(* IEC 61131-3 sources: RAG_PLC/data/result/test/022, 2 files *)

(* ---- wrapped.st ---- *)
(* =========================================================
   Generated by PLC-Eval Benchmark Wrapper
   ========================================================= *)

FUNCTION_BLOCK LLM_Wrapper_FB
PROGRAM Main
VAR
    StartChk : BOOL;
    Regen : BOOL;
    ErrorFlag : BOOL;
END_VAR

// Step 1: Start Check
IF NOT StartChk THEN
    StartChk := TRUE;
    // Additional initialization code here
END_IF;

// Step 2: Regeneration Check
IF StartChk AND NOT Regen THEN
    Regen := TRUE;
    // Additional regeneration code here
END_IF;

// Error Handling
IF ErrorFlag THEN
    // Stop program
    // Issue error message to visualization system
    // Additional error handling code here
END_IF;

END_PROGRAM
END_FUNCTION_BLOCK

PROGRAM Auto_Proxy_Prg
  VAR
    instance : LLM_Wrapper_FB;
  END_VAR

  instance();
END_PROGRAM

CONFIGURATION Config0
  RESOURCE Res0 ON PLC
    TASK TaskMain(INTERVAL := T#20ms, PRIORITY := 0);
    PROGRAM Inst0 WITH TaskMain : Auto_Proxy_Prg;
  END_RESOURCE
END_CONFIGURATION

(* ---- raw_code.st ---- *)
PROGRAM Main
VAR
    StartChk : BOOL;
    Regen : BOOL;
    ErrorFlag : BOOL;
END_VAR

// Step 1: Start Check
IF NOT StartChk THEN
    StartChk := TRUE;
    // Additional initialization code here
END_IF;

// Step 2: Regeneration Check
IF StartChk AND NOT Regen THEN
    Regen := TRUE;
    // Additional regeneration code here
END_IF;

// Error Handling
IF ErrorFlag THEN
    // Stop program
    // Issue error message to visualization system
    // Additional error handling code here
END_IF;

END_PROGRAM
